// TIA Portal project "bottel line" (V16)
// Vorlageprojekt für das Buch mit Zielsystem S7-1200

(* hardware
DEVICE "S7-1200-Station_1"  S7-1200 Station
   slot 0: "Baugruppenträger_0"  Rack  V1.0
   slot 1: "PLC_1"  CPU 1211C DC/DC/DC  6ES7 211-1AE40-0XB0  V4.1
*)

// ===== PLC "PLC_1"  CPU 1211C DC/DC/DC =====

VAR_GLOBAL   // PLC tag table "Standard-Variablentabelle"
   "start" AT %I0.0 : Bool;
   "stop" AT %I0.1 : Bool;
   "x1" AT %M0.0 : Bool;
   "fill valve" AT %Q0.0 : Bool;
   "x2" AT %M0.1 : Bool;
   "y6" AT %M0.7 : Bool;
   "y1" AT %M0.2 : Bool;
   "place 1z" AT %Q0.2 : Bool;
   "x3" AT %M0.3 : Bool;
   "s" AT %I0.2 : Bool;
   "y4" AT %M0.6 : Bool;
   "y3" AT %M0.5 : Bool;
   "discharge valve" AT %Q0.1 : Bool;
   "y2" AT %M0.4 : Bool;
   "4m" AT %Q0.3 : Bool;
END_VAR

// folder: System blocks/Program resources

DATA_BLOCK "T1"   // DB1
{ S7_Optimized_Access := 'TRUE' }
AUTHOR : Simatic
FAMILY : IEC
NAME : IEC_TMR
VERSION : 1.0
// stored: InstanceOfName IEC_TIMER
"IEC_TIMER"
BEGIN
END_DATA_BLOCK

DATA_BLOCK "T2"   // DB2
{ S7_Optimized_Access := 'TRUE' }
AUTHOR : Simatic
FAMILY : IEC
NAME : IEC_TMR
VERSION : 1.0
// stored: InstanceOfName IEC_TIMER
"IEC_TIMER"
BEGIN
END_DATA_BLOCK

DATA_BLOCK "T3"   // DB3
{ S7_Optimized_Access := 'TRUE' }
AUTHOR : Simatic
FAMILY : IEC
NAME : IEC_TMR
VERSION : 1.0
// stored: InstanceOfName IEC_TIMER
"IEC_TIMER"
BEGIN
END_DATA_BLOCK

DATA_BLOCK "C1"   // DB4
{ S7_Optimized_Access := 'TRUE' }
AUTHOR : Simatic
FAMILY : IEC
NAME : CNTR
VERSION : 1.0
// stored: InstanceOfName IEC_COUNTER
"IEC_COUNTER"
BEGIN
END_DATA_BLOCK

// folder: (top level)

FUNCTION "MHJ-PLC-Lab-Function-S71200" : Void   // FC9000, SCL
{ S7_Optimized_Access := 'TRUE' }
VERSION : 0.1
   VAR_TEMP
      rdTimeReturn : Int;
      outputTime : DTL;
      SyncVal : Byte;
      forVal : Int;
      forVal_2 : Int;
      Value : Byte;
   END_VAR
   VAR CONSTANT
      CompVal : Byte := 16#34;
      Value_01 : Byte := 16#11;
      Value_01_DW : DWord := 16#A165_D992;
      Value_02_DW : DWord := 16#58BE_4401;
   END_VAR
BEGIN

   #Value:=PEEK(area := 16#82,
        dbNumber := 0,
        byteOffset := 511);
   #Value := #Value + 1;

   POKE(area := 16#82,
        dbNumber := 0,
        byteOffset := 511,
        value := #Value);

   POKE(area:=16#81,
        dbNumber:=0,
        byteOffset:=1016,
        value:=#Value_01_DW);
   POKE(area := 16#81,
        dbNumber := 0,
        byteOffset := 1020,
        value := #Value_02_DW);

   POKE(area := 16#81,
        dbNumber := 0,
        byteOffset := 511,
        value := B#16#00);

   FOR #forVal := 0 TO 120 DO
       FOR #forVal_2:=0 TO 10 DO
           #rdTimeReturn:=RD_SYS_T(#outputTime);
           #rdTimeReturn := WR_SYS_T(#outputTime);
           #rdTimeReturn := RD_SYS_T(#outputTime);
           #rdTimeReturn := WR_SYS_T(#outputTime);
       END_FOR;
       #SyncVal:= PEEK(area := 16#81,
                      dbNumber := 0,
                      byteOffset := 511);
       IF #SyncVal = #CompVal THEN
          GOTO M_1;
       END_IF;
   END_FOR;
   RETURN;

   M_1:
   POKE(area := 16#81,
        dbNumber := 0,
        byteOffset := 511,
        value := B#16#0);
END_FUNCTION

ORGANIZATION_BLOCK "Main"   // OB1, LAD, ProgramCycle
TITLE = "Main Program Sweep (Cycle)"
{ S7_Optimized_Access := 'TRUE' }
VERSION : 0.1
   VAR_INPUT
      Initial_Call : Bool;   // Initial call of this OB
      Remanence : Bool;   // =True, if remanent data are available
   END_VAR
BEGIN

REGION Network 1: Konnektierungsbaustein für PLC-Lab
   // Im Netzwerk 1 wird der Konnektierungsbaustein für PLC-Lab aufgerufen.
   // Dieser Aufruf darf nicht entfernt werden!
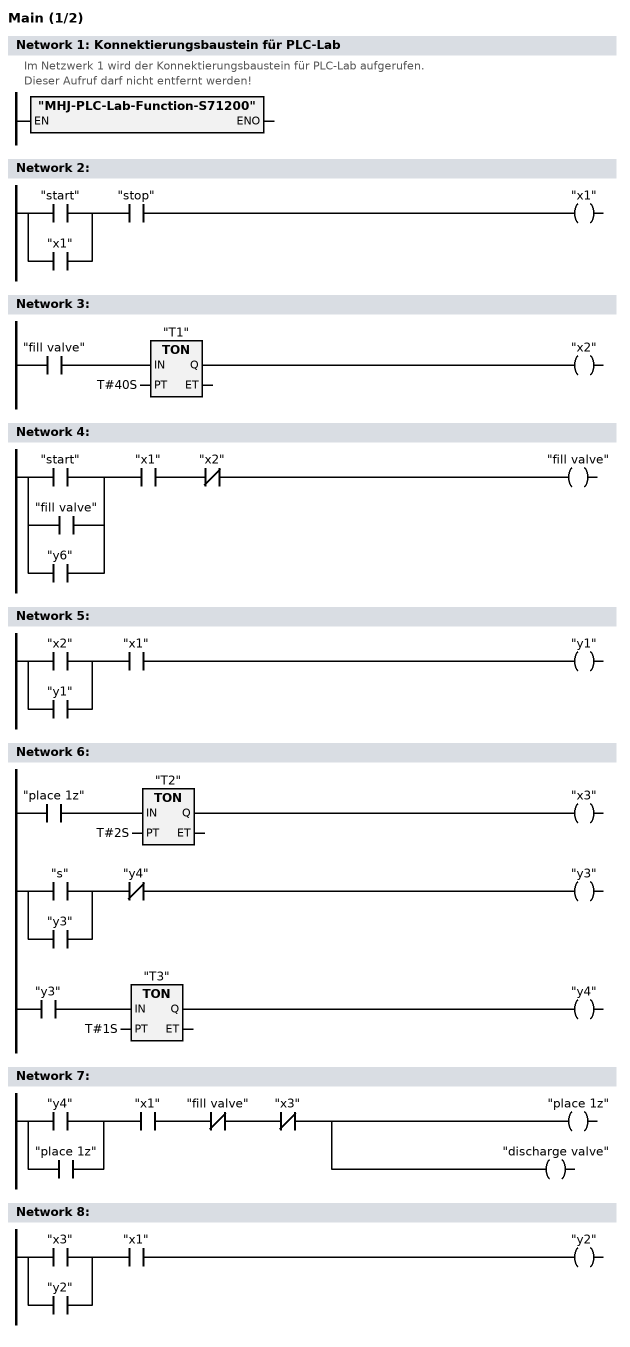
   RUNG wire#powerrail
      "MHJ-PLC-Lab-Function-S71200"()
   END_RUNG
   // the same network as SCL:
   "MHJ-PLC-Lab-Function-S71200"();
END_REGION

REGION Network 2
   RUNG wire#powerrail
      Contact( "start" )
      wire#w1
      Contact( "stop" )
      Coil( "x1" )
   END_RUNG
   RUNG wire#powerrail
      Contact( "x1" )
   END_RUNG wire#w1
   // the same network as SCL:
   "x1" := ("start" OR "x1") AND "stop";
END_REGION

REGION Network 3
   "T1".TON(IN := "fill valve", PT := T#40S);
   "x2" := "T1".Q;
END_REGION

REGION Network 4
   RUNG wire#powerrail
      Contact( "start" )
      wire#w1
      Contact( "x1" )
      I_Contact( "x2" )
      Coil( "fill valve" )
   END_RUNG
   RUNG wire#powerrail
      Contact( "fill valve" )
   END_RUNG wire#w1
   RUNG wire#powerrail
      Contact( "y6" )
   END_RUNG wire#w1
   // the same network as SCL:
   "fill valve" := ("start" OR "fill valve" OR "y6") AND "x1" AND NOT "x2";
END_REGION

REGION Network 5
   RUNG wire#powerrail
      Contact( "x2" )
      wire#w1
      Contact( "x1" )
      Coil( "y1" )
   END_RUNG
   RUNG wire#powerrail
      Contact( "y1" )
   END_RUNG wire#w1
   // the same network as SCL:
   "y1" := ("x2" OR "y1") AND "x1";
END_REGION

REGION Network 6
   "T2".TON(IN := "place 1z", PT := T#2S);
   "x3" := "T2".Q;
   "y3" := ("s" OR "y3") AND NOT "y4";
   "T3".TON(IN := "y3", PT := T#1S);
   "y4" := "T3".Q;
END_REGION

REGION Network 7
   RUNG wire#powerrail
      Contact( "y4" )
      wire#w1
      Contact( "x1" )
      I_Contact( "fill valve" )
      I_Contact( "x3" )
      wire#w2
      Coil( "place 1z" )
   END_RUNG
   RUNG wire#powerrail
      Contact( "place 1z" )
   END_RUNG wire#w1
   RUNG wire#w2
      Coil( "discharge valve" )
   END_RUNG
   // the same network as SCL:
   "place 1z" := ("y4" OR "place 1z") AND "x1" AND NOT "fill valve" AND NOT "x3";
   "discharge valve" := "place 1z";
END_REGION

REGION Network 8
   RUNG wire#powerrail
      Contact( "x3" )
      wire#w1
      Contact( "x1" )
      Coil( "y2" )
   END_RUNG
   RUNG wire#powerrail
      Contact( "y2" )
   END_RUNG wire#w1
   // the same network as SCL:
   "y2" := ("x3" OR "y2") AND "x1";
END_REGION

REGION Network 9
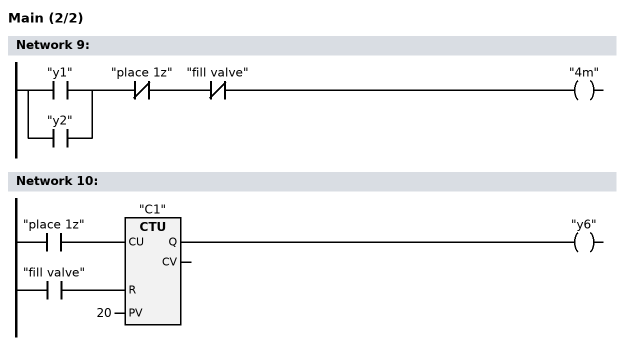
   RUNG wire#powerrail
      Contact( "y1" )
      wire#w1
      I_Contact( "place 1z" )
      I_Contact( "fill valve" )
      Coil( "4m" )
   END_RUNG
   RUNG wire#powerrail
      Contact( "y2" )
   END_RUNG wire#w1
   // the same network as SCL:
   "4m" := ("y1" OR "y2") AND NOT "place 1z" AND NOT "fill valve";
END_REGION

REGION Network 10
   "C1".CTU(CU := "place 1z", R := "fill valve", PV := 20);
   "y6" := "C1".Q;
END_REGION
END_ORGANIZATION_BLOCK